// TIA Portal V17 export
// export: Created 2025-03-05T08:01:41.2210901Z, ExportSetting WithDefaults, DisplayName Totally Integrated Automation Portal, DisplayVersion V17 Update 8, DisplayName TIA Portal Openness, DisplayVersion V17 Update 8, DisplayName TIA Portal Version Control Interface, DisplayVersion V17, DisplayName SINAMICS Startdrive Advanced, DisplayVersion V17 SP2, DisplayName SINAMICS Startdrive G110M, G120, G120C, G120D, G120P, G115D, DisplayVersion V17 SP2, DisplayName SINAMICS Startdrive G130, G150, S120, S150, SINAMICS MV, S210, DisplayVersion V17 SP2, DisplayName STEP 7 Professional, DisplayVersion V17 Update 8, DisplayName SINUMERIK ONE STEP 7 Toolbox, DisplayVersion V17 Update 12, DisplayName SINUMERIK 840D sl STEP 7 Toolbox, DisplayVersion V17 Update 12, DisplayName STEP 7 Safety, DisplayVersion V17 Update 6, DisplayName WinCC Advanced, DisplayVersion V17 Update 8
FUNCTION "FC7227_24_HOURS_TEST" : Void   // FC7227, LAD
{ S7_Optimized_Access := 'FALSE' }
AUTHOR : ETXETAR
VERSION : 1.0
// stored: AutoNumber false, IsIECCheckEnabled false, SetENOAutomatically false, UDAEnableTagReadback false
   VAR_TEMP
      ERROR1 : Int;
      DataTime : Date_And_Time;
      T1 : Bool;
   END_VAR
   VAR CONSTANT
      FC_NUMBER : DInt := 7227;
   END_VAR
   VAR_TEMP   // added for the SCL form of the ladder/FBD networks
      _w1 : Bool;
   END_VAR
BEGIN

REGION Network 1: TEST 24H START REQ AUX
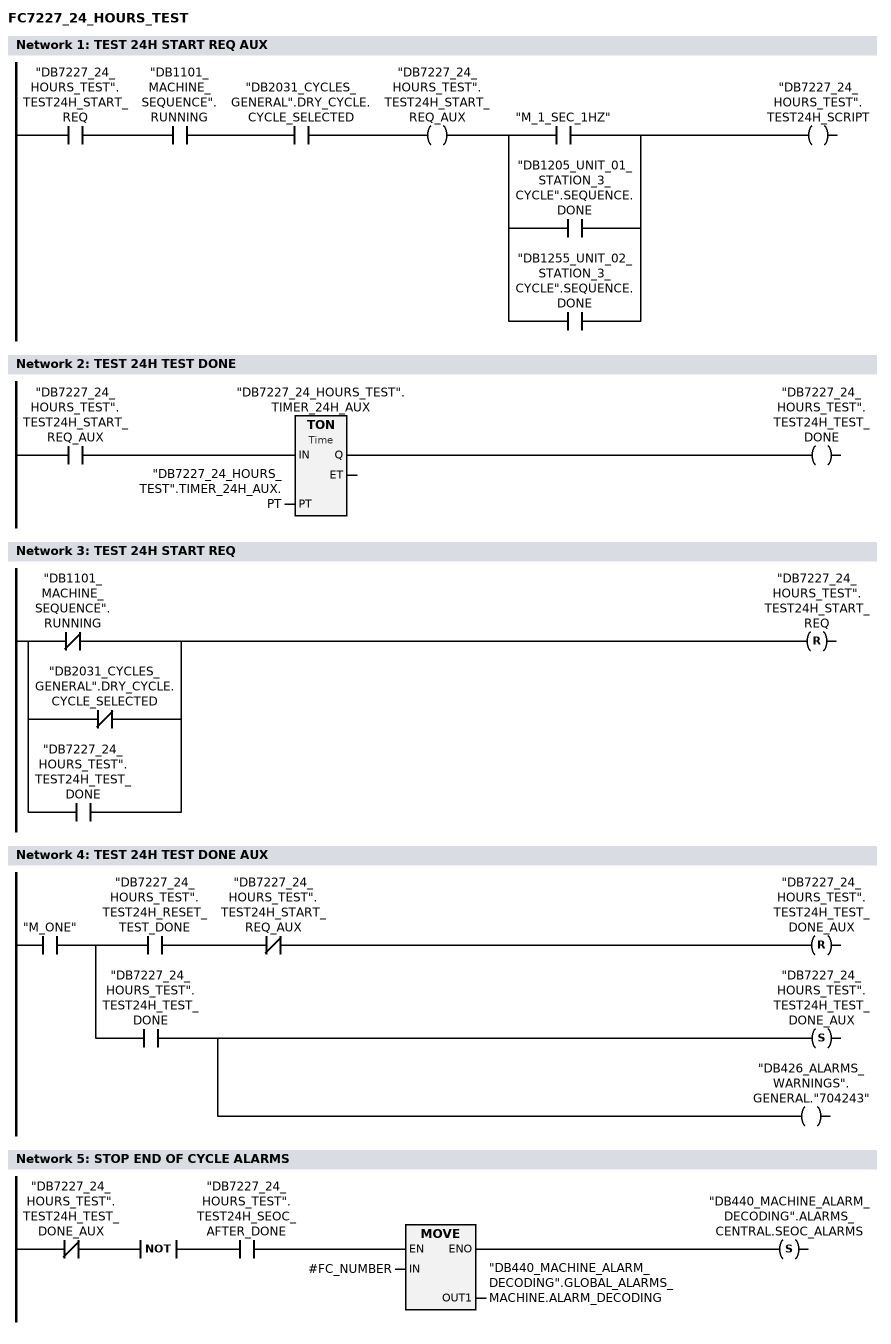
   RUNG wire#powerrail
      Contact( "DB7227_24_HOURS_TEST".TEST24H_START_REQ )
      Contact( "DB1101_MACHINE_SEQUENCE".RUNNING )
      Contact( "DB2031_CYCLES_GENERAL".DRY_CYCLE.CYCLE_SELECTED )
      Coil( "DB7227_24_HOURS_TEST".TEST24H_START_REQ_AUX )
      wire#w1
      Contact( "M_1_SEC_1HZ" )
      wire#w2
      Coil( "DB7227_24_HOURS_TEST".TEST24H_SCRIPT )
   END_RUNG
   RUNG wire#w1
      Contact( "DB1205_UNIT_01_STATION_3_CYCLE".SEQUENCE.DONE )
   END_RUNG wire#w2
   RUNG wire#w1
      Contact( "DB1255_UNIT_02_STATION_3_CYCLE".SEQUENCE.DONE )
   END_RUNG wire#w2
   // the same network as SCL:
   "DB7227_24_HOURS_TEST".TEST24H_START_REQ_AUX := "DB7227_24_HOURS_TEST".TEST24H_START_REQ AND "DB1101_MACHINE_SEQUENCE".RUNNING AND "DB2031_CYCLES_GENERAL".DRY_CYCLE.CYCLE_SELECTED;
   "DB7227_24_HOURS_TEST".TEST24H_SCRIPT := "DB7227_24_HOURS_TEST".TEST24H_START_REQ_AUX AND ("M_1_SEC_1HZ" OR "DB1205_UNIT_01_STATION_3_CYCLE".SEQUENCE.DONE OR "DB1255_UNIT_02_STATION_3_CYCLE".SEQUENCE.DONE);
END_REGION

REGION Network 2: TEST 24H TEST DONE
   RUNG wire#powerrail
      Contact( "DB7227_24_HOURS_TEST".TEST24H_START_REQ_AUX )
      { S7_Templates := "time_type := Time" } "DB7227_24_HOURS_TEST".TIMER_24H_AUX.TON(pt := "DB7227_24_HOURS_TEST".TIMER_24H_AUX.PT, et =>)
      Coil( "DB7227_24_HOURS_TEST".TEST24H_TEST_DONE )
   END_RUNG
   // the same network as SCL:
   "DB7227_24_HOURS_TEST".TIMER_24H_AUX.TON(IN := "DB7227_24_HOURS_TEST".TEST24H_START_REQ_AUX,
                           PT := "DB7227_24_HOURS_TEST".TIMER_24H_AUX.PT);
   "DB7227_24_HOURS_TEST".TEST24H_TEST_DONE := "DB7227_24_HOURS_TEST".TIMER_24H_AUX.Q;
END_REGION

REGION Network 3: TEST 24H START REQ
   RUNG wire#powerrail
      I_Contact( "DB1101_MACHINE_SEQUENCE".RUNNING )
      wire#w1
      R_Coil( "DB7227_24_HOURS_TEST".TEST24H_START_REQ )
   END_RUNG
   RUNG wire#powerrail
      I_Contact( "DB2031_CYCLES_GENERAL".DRY_CYCLE.CYCLE_SELECTED )
   END_RUNG wire#w1
   RUNG wire#powerrail
      Contact( "DB7227_24_HOURS_TEST".TEST24H_TEST_DONE )
   END_RUNG wire#w1
   // the same network as SCL:
   IF NOT "DB1101_MACHINE_SEQUENCE".RUNNING OR NOT "DB2031_CYCLES_GENERAL".DRY_CYCLE.CYCLE_SELECTED OR "DB7227_24_HOURS_TEST".TEST24H_TEST_DONE THEN
       "DB7227_24_HOURS_TEST".TEST24H_START_REQ := FALSE;
   END_IF;
END_REGION

REGION Network 4: TEST 24H TEST DONE AUX
   RUNG wire#powerrail
      Contact( "M_ONE" )
      wire#w1
      Contact( "DB7227_24_HOURS_TEST".TEST24H_RESET_TEST_DONE )
      I_Contact( "DB7227_24_HOURS_TEST".TEST24H_START_REQ_AUX )
      R_Coil( "DB7227_24_HOURS_TEST".TEST24H_TEST_DONE_AUX )
   END_RUNG
   RUNG wire#w1
      Contact( "DB7227_24_HOURS_TEST".TEST24H_TEST_DONE )
      wire#w2
      S_Coil( "DB7227_24_HOURS_TEST".TEST24H_TEST_DONE_AUX )
   END_RUNG
   RUNG wire#w2
      Coil( "DB426_ALARMS_WARNINGS".GENERAL."704243" )
   END_RUNG
   // the same network as SCL:
   IF "M_ONE" AND "DB7227_24_HOURS_TEST".TEST24H_RESET_TEST_DONE AND NOT "DB7227_24_HOURS_TEST".TEST24H_START_REQ_AUX THEN
       "DB7227_24_HOURS_TEST".TEST24H_TEST_DONE_AUX := FALSE;
   END_IF;
   #_w1 := "M_ONE" AND "DB7227_24_HOURS_TEST".TEST24H_TEST_DONE;
   IF #_w1 THEN "DB7227_24_HOURS_TEST".TEST24H_TEST_DONE_AUX := TRUE; END_IF;
   "DB426_ALARMS_WARNINGS".GENERAL."704243" := #_w1;
END_REGION

REGION Network 5: STOP END OF CYCLE ALARMS
   RUNG wire#powerrail
      I_Contact( "DB7227_24_HOURS_TEST".TEST24H_TEST_DONE_AUX )
      Not()
      Contact( "DB7227_24_HOURS_TEST".TEST24H_SEOC_AFTER_DONE )
      { S7_GenerateENO := "TRUE" } Move(in := #FC_NUMBER, out1 => "DB440_MACHINE_ALARM_DECODING".GLOBAL_ALARMS_MACHINE.ALARM_DECODING)
      S_Coil( "DB440_MACHINE_ALARM_DECODING".ALARMS_CENTRAL.SEOC_ALARMS )
   END_RUNG
   // the same network as SCL:
   // ENO of a box is taken as its EN; it also drops when the box reports an error
   IF NOT (NOT "DB7227_24_HOURS_TEST".TEST24H_TEST_DONE_AUX) AND "DB7227_24_HOURS_TEST".TEST24H_SEOC_AFTER_DONE THEN
       "DB440_MACHINE_ALARM_DECODING".GLOBAL_ALARMS_MACHINE.ALARM_DECODING := #FC_NUMBER;
       "DB440_MACHINE_ALARM_DECODING".ALARMS_CENTRAL.SEOC_ALARMS := TRUE;
   END_IF;
END_REGION

NETWORK
TITLE = READ TIME
      CALL  RD_SYS_T
      ( RET_VAL := #ERROR1,
        OUT     := #DataTime
      );
      LAR1  P##DataTime;
      L     B [AR1, P#0.0];
      BTI;
      T     "DB7227_24_HOURS_TEST".TEMP_DATA.Year;
      L     B [AR1, P#1.0];
      BTI;
      T     "DB7227_24_HOURS_TEST".TEMP_DATA.Month;
      L     B [AR1, P#2.0];
      BTI;
      T     "DB7227_24_HOURS_TEST".TEMP_DATA.Day;
      L     B [AR1, P#3.0];
      BTI;
      T     "DB7227_24_HOURS_TEST".TEMP_DATA.Hour;
      L     B [AR1, P#4.0];
      BTI;
      T     "DB7227_24_HOURS_TEST".TEMP_DATA.Minute;
      L     B [AR1, P#5.0];
      BTI;
      T     "DB7227_24_HOURS_TEST".TEMP_DATA.Second;

END_FUNCTION
